TYPE (* IEC61131-3, Table 14#5 *)
  (* Standard: 1131-3 *)
  (* Version 0.0, 1/8/2024, Cheyan, Schneider Electric, Template *)
  PACKAGE Main;
  {SET_ATTRIBUTE(nxtDataType, QdpEwqSPB7qJkv5aCelDKTYtUgsad/yJ+BPQSBlH6p5whmzrBuOANBbyK94d3S89KrvA7rF1kXXxVvHbrHnKvM8bXkItqItpPUwT2tXHh1fYow+RByLcBFo546BnFZoBpIpMpJ45yJne+/kXj2+ugTuygtvdG5jJm+9zuCx6ys3rXg7S1fgYVV+sPWsFq9L1)}
  TimeStamp : STRUCT
    SecondSinceEpoch : UDINT;
    FractionOfSecond : UDINT;
    TimeQuality : TimeQuality;
  END_STRUCT;
END_TYPE
